// TIA Portal V19 export
DATA_BLOCK "Mémoires"   // DB2
   VAR RETAIN
      "Mode Manuel" : Bool;
      "Affichage hauteur" : Int;
      "HMI BP Ascenceur Haut" : Bool;
      "HMI BP Ascenceur Bas" : Bool;
      "HMI BP Ejection" : Bool;
      "HMI SW Glissière" : Bool;
      "Erreur Montée Ascenceur" : Int;
      "Erreur Descente Ascenceur" : Int;
      "Erreur Ejection" : Int;
      "Erreur Capteurs" : Int;
   END_VAR
BEGIN
END_DATA_BLOCK
